Fanuc KAREL source: kb00081.KL

-- PROVISIONAL review KL for V940-1; original PC SHA256 908a23cf3c4ec188d4b35cb6577daddc79d3cce93eee7a1519b27cdc68e03666
-- Incomplete behavior may be omitted. Consult companion uncertainty JSON. Do not deploy.
PROGRAM KB00081
%NOLOCKGROUP
BEGIN
  -- V9_ZERO_TABLE_METADATA_HINT layout=0002_ascii; no indexed target words; source/name/runtime held
  -- UNRESOLVED_PC offsets 5-12; opcodes 9D,23
  -- UNRESOLVED_PC offsets 17-24; opcodes 9D,23
  -- UNRESOLVED_PC offsets 29-36; opcodes 9D,23
  -- UNRESOLVED_PC offsets 41-69; opcodes 27,22,22,22,31,23
  -- UNRESOLVED_PC offsets 74-78; opcodes 7F
END KB00081
